(* PLC project logical_or_10, Dassault Systèmes ControlBuild 2024x *)
(* stored: creationDateTime 2023-10-03T11:13:28-01:00 *)

(* This module makes a "logical OR" operation between inputs. Number of inputs can go from 2 to 10. Result is a boolean. *)
FUNCTION_BLOCK equipment_library.logical_or_10
  VAR_INPUT
    inputBit1 : BOOL := false;
    inputBit2 : BOOL := false;
    inputBit3 : BOOL := false;
    inputBit4 : BOOL := false;
    inputBit5 : BOOL := false;
    inputBit6 : BOOL := false;
    inputBit7 : BOOL := false;
    inputBit8 : BOOL := false;
    inputBit9 : BOOL := false;
    inputBit10 : BOOL := false;
  END_VAR
  VAR_OUTPUT
    outputBit : BOOL := false;
  END_VAR
  VAR CONSTANT
    input1Logic : BOOL := true;
    input2Logic : BOOL := true;
    input3Logic : BOOL := true;
    input4Logic : BOOL := true;
    input5Logic : BOOL := true;
    input6Logic : BOOL := true;
    input7Logic : BOOL := true;
    input8Logic : BOOL := true;
    input9Logic : BOOL := true;
    input10Logic : BOOL := true;
    outputLogic : BOOL := true;
    nbInputs : DINT := 10;
  END_VAR
  VAR
    d_output : BOOL := false;
    v_d_output : BOOL := true;
  END_VAR


ACTION C_source_code:
/* ----------------------------------------------------------------	*/
/* Type : Model of Operative Behaviour					*/
/* Category :  Toolbox							*/
/* Author : Dassault Systemes						*/
/* Update date : June 2018						*/
/* ----------------------------------------------------------------	*/
/* This module makes a "logical OR" operation between inputs. 	*/
/* Number of inputs can gone from 2 to 10. 				*/
/* Number of inputs is given by the nbInputs parameter.		*/
/* Result is a boolean.							*/
/* The output can be preset	by the user					*/
/* ----------------------------------------------------------------	*/

/* Declaration area of temporary variables */

CB_Bool inputsArray[11];
CB_Bool logicArray[11];
CB_Int index;



if (d_output|| (nbInputs<2) || (nbInputs>10)) outputBit=v_d_output;
else  {
	inputsArray[0]=inputBit1; logicArray[0]=input1Logic;
	inputsArray[1]=inputBit2; logicArray[1]=input2Logic;
	inputsArray[2]=inputBit3; logicArray[2]=input3Logic;
	inputsArray[3]=inputBit4; logicArray[3]=input4Logic;
	inputsArray[4]=inputBit5; logicArray[4]=input5Logic;
	inputsArray[5]=inputBit6; logicArray[5]=input6Logic;
	inputsArray[6]=inputBit7; logicArray[6]=input7Logic;
	inputsArray[7]=inputBit8; logicArray[7]=input8Logic;
	inputsArray[8]=inputBit9; logicArray[8]=input9Logic;
	inputsArray[9]=inputBit10; logicArray[9]=input10Logic;
	outputBit = 0;
	for (index=0;index<nbInputs;index++)
		outputBit = outputBit | (inputsArray[index] ^ ! logicArray[index]);
	outputBit = outputBit ^ ! outputLogic;
}
END_ACTION
END_FUNCTION_BLOCK
